{attribute 'GeneratedUsingTerminal: EL9540--0000'}
{attribute addProperty BoxType "EL9540--0000"}
{attribute addProperty Description "EL9540 Surge/Overvoltagefilter (Power supply)"}
{attribute addProperty Physics "KK"}
{attribute addProperty Id "EL9540"}
{attribute addProperty CRC "1125899883"}
{attribute addProperty Size "0"}
TYPE EL9540_431BDE6B EXTENDS EtcSlaveTerminalBase_947E5A46 :
STRUCT
END_STRUCT
END_TYPE

(* stored: Version 1.2.0.0, ProductVersion 3.1.4024.9
   DUT EL9540_431BDE6B: Id {d009e989-2339-40dd-8f11-760553a56105} *)
